(* Logix 5000 project; controller ProyectoIntegrador Emulate 5570 rev 30.12; software revision 30.00 *)

TASK MainTask (continuous, watchdog 500 ms) : MainProgram

MODULES
   Local : Emulate 5570 (ICP 2, rev 30.12)
      IO_module : vendor 1 type 0 code 15 (ICP 3, rev 1.1, Output RPI 150 ms)
END_MODULES

PROGRAM MainProgram   (* main routine MainRoutine *)
VAR
   Action_000 : SFC_ACTION := (Status := 16#0020_0000, PauseTimer := 1);
   Action_001 : SFC_ACTION := (Status := 16#0020_0000, PauseTimer := 1);
   Action_002 : SFC_ACTION := (Status := 16#0020_0000, PauseTimer := 1);
   Action_003 : SFC_ACTION := (Status := 16#0020_0000, PauseTimer := 1);
   Action_004 : SFC_ACTION := (Status := 16#0020_0000, PauseTimer := 1);
   Action_005 : SFC_ACTION := (Status := 16#0020_0000, PauseTimer := 1);
   Action_006 : SFC_ACTION := (Status := 16#0020_0000, PauseTimer := 1);
   Action_007 : SFC_ACTION := (Status := 16#0020_0000, PauseTimer := 1);
   Action_008 : SFC_ACTION := (Status := 16#0020_0000, PauseTimer := 1);
   Action_009 : SFC_ACTION := (Status := 16#0020_0000, PauseTimer := 1);
   Action_010 : SFC_ACTION := (Status := 16#0020_0000, PauseTimer := 1);
   Action_011 : SFC_ACTION := (Status := 16#0020_0000, PauseTimer := 1);
   Action_012 : SFC_ACTION := (Status := 16#0020_0000, PauseTimer := 1);
   Action_013 : SFC_ACTION := (Status := 16#0020_0000, PauseTimer := 1);
   Action_014 : SFC_ACTION := (Status := 16#0020_0000, PauseTimer := 1);
   Action_015 : SFC_ACTION := (Status := 16#0020_0000, PauseTimer := 1);
   Action_016 : SFC_ACTION := (Status := 16#0020_0000, PauseTimer := 1);
   Action_017 : SFC_ACTION := (Status := 16#0020_0000, PauseTimer := 1);
   Action_018 : SFC_ACTION := (Status := 16#0020_0000, PauseTimer := 1);
   Action_019 : SFC_ACTION := (Status := 16#0020_0000, PauseTimer := 1);
   Action_020 : SFC_ACTION := (Status := 16#0020_0000, PauseTimer := 1);
   Action_021 : SFC_ACTION := (Status := 16#0020_0000, PauseTimer := 1);
   Action_022 : SFC_ACTION := (Status := 16#0020_0000, PauseTimer := 1);
   Action_023 : SFC_ACTION := (Status := 16#0020_0000, PauseTimer := 1);
   Action_024 : SFC_ACTION := (Status := 16#0020_0000, PauseTimer := 1);
   Action_025 : SFC_ACTION := (Status := 16#0020_0000, PauseTimer := 1);
   Action_026 : SFC_ACTION := (Status := 16#0020_0000, PauseTimer := 1);
   Action_027 : SFC_ACTION := (Status := 16#0020_0000, PauseTimer := 1);
   Action_028 : SFC_ACTION := (Status := 16#0020_0000, PauseTimer := 1);
   Action_029 : SFC_ACTION := (Status := 16#0020_0000, PauseTimer := 1);
   BC_1 : BOOL;   // Encender/Apagar conveyor belt 1
   BC_2 : BOOL;   // Encender/Apagar conveyor belt 2
   BC_3 : BOOL;   // Encender/Apagar conveyor belt 3
   C1b : BOOL;   // Moves Cilinder 1 backward
   C1f : BOOL;   // Move cilinder 1 forward
   C2b : DINT;   // Move the cilinder 2 backwards
   C2f : BOOL;   // Move the cilinder 2 forward
   Cinta_gra : BOOL;   // El robot ya pegado en las cajas de la cinta grande
   Cinta_med : BOOL;   // El robot ya pegado en las cajas de la cinta media
   CintaRob : BOOL;   // El robot ya pegado en las cajas de la cinta pequena
   Clasif : BOOL;   // Encender/Apagar Classificador
   Compressor : BOOL;   // Encender/Apagar Compressor
   cont1 : COUNTER := (PRE := 3);
   cont2 : COUNTER := (PRE := 3);
   cont3 : COUNTER := (PRE := 3);
   cont4 : COUNTER := (PRE := 3);
   cont5 : COUNTER := (PRE := 3);
   cont6 : COUNTER := (PRE := 3);
   isBlue : BOOL;   // If the color detector in front of cilinder 1 detects blue color
   isGreen : BOOL;   // If the color detector in front of cilinder 1 detects green color
   isRed : BOOL;   // Normal or Color sensor for big boxes
   K1 : BOOL;   // Move la banda trasnportadora para esquerda y para trás
   K2 : BOOL;   // Move la banda transportadora para la direcha y para adelante
   K3 : BOOL;   // Move la banda trasnportadora para esquerda y para trás
   K4 : BOOL;   // Move la banda transportadora para la direcha y para adelante
   K5 : BOOL;   // Move la banda trasnportadora para esquerda y para trás
   K6 : BOOL;   // Move la banda transportadora para la direcha y para adelante
   Lavdo : BOOL;   // Encender/Apagar Lavado
   lConv : BOOL;   // Sensor de cajas conveyor belt 3 (vegetal grande)
   lCount : DINT;   // Large box counter
   mConv : BOOL;
   mCount : DINT;   // Medium Boxes count
   RC5 : BOOL;   // Encender/Apagar roller conveyor 4
   RC_1 : BOOL;   // Encender/Apagar roller conveyor 1
   RC_2 : BOOL;   // Encender/Apagar roller conveyor 2
   RC_3 : BOOL;   // Encender/Apagar roller conveyor 3
   RC_4 : BOOL;   // Encender/Apagar roller conveyor 4
   robotReady_L : BOOL;   // Un nível esta listo en la banda de cajas grandes
   robotReady_M : BOOL;   // Un nível esta listo en la banda de cajas medias
   robotReady_S : BOOL;   // Un nível esta listo en la banda de cajas pequenas
   S1_C1 : BOOL;   // Cilindro 1 recogido
   S1_C2 : BOOL;   // Sensor 1 final de carrera cilindro2
   S2_C1 : BOOL;   // Sensor 2 final de carrera cilindro 1
   S2_C2 : BOOL;   // Sensor 2 final de carrera cilindro 2
   S_clasif : DINT;   // Sensor para clasificacion de empaque
   sBC1 : BOOL;   // Tenemos una caja en el fin del tapete BC1
   sBC2 : BOOL;   // Tenemos una caja en el fin del tapete BC2
   sBC3 : BOOL;   // Tenemos una caja en el fin del tapete BC3
   sCount : DINT;   // Small Boxes Count
   Secado : BOOL;   // Encender/Apagar Secado
   Start : BOOL;   // Inicio del proceso
   Step_000 : SFC_STEP := (Status := 16#a820_0201, X := 1, SA := 1, DN := 1, PauseTimer := 1, T := 1176385, TMax := 1176385, Count := 1);
   Step_001 : SFC_STEP := (Status := 16#0020_0000, PauseTimer := 1);
   Step_002 : SFC_STEP := (Status := 16#0020_0000, PauseTimer := 1);
   Step_003 : SFC_STEP := (Status := 16#0020_0000, PauseTimer := 1);
   Step_004 : SFC_STEP := (Status := 16#0020_0000, PauseTimer := 1);
   Step_005 : SFC_STEP := (Status := 16#0020_0000, PauseTimer := 1);
   Step_006 : SFC_STEP := (Status := 16#0020_0000, PauseTimer := 1);
   Step_007 : SFC_STEP := (Status := 16#0020_0000, PauseTimer := 1);
   Step_008 : SFC_STEP := (Status := 16#0020_0000, PauseTimer := 1);
   Step_009 : SFC_STEP := (Status := 16#0020_0000, PauseTimer := 1);
   Step_010 : SFC_STEP := (Status := 16#0020_0000, PauseTimer := 1);
   Step_011 : SFC_STEP := (Status := 16#0020_0001, PauseTimer := 1);
   Step_012 : SFC_STEP := (Status := 16#0020_0001, PauseTimer := 1);
   Step_013 : SFC_STEP := (Status := 16#0020_0001, PauseTimer := 1);
   Step_014 : SFC_STEP := (Status := 16#0020_0001, PauseTimer := 1);
   Step_015 : SFC_STEP := (Status := 16#0020_0001, PauseTimer := 1);
   Step_016 : SFC_STEP := (Status := 16#0020_0000, PauseTimer := 1);
   Step_017 : SFC_STEP := (Status := 16#0020_0000, PauseTimer := 1);
   Step_018 : SFC_STEP := (Status := 16#0020_0000, PauseTimer := 1);
   Step_019 : SFC_STEP := (Status := 16#0020_0000, PauseTimer := 1);
   Step_020 : SFC_STEP := (Status := 16#0020_0000, PauseTimer := 1);
   Step_021 : SFC_STEP := (Status := 16#0020_0001, PauseTimer := 1);
   Step_022 : SFC_STEP := (Status := 16#0020_0001, PauseTimer := 1);
   Step_023 : SFC_STEP := (Status := 16#0020_0001, PauseTimer := 1);
   Step_024 : SFC_STEP := (Status := 16#0020_0001, PauseTimer := 1);
   Step_025 : SFC_STEP := (Status := 16#0020_0001, PauseTimer := 1);
   Step_026 : SFC_STEP := (Status := 16#0020_0000, PauseTimer := 1);
   Step_027 : SFC_STEP := (Status := 16#0020_0000, PauseTimer := 1);
   Step_028 : SFC_STEP := (Status := 16#0020_0000, PauseTimer := 1);
   Step_029 : SFC_STEP := (Status := 16#0020_0000, PauseTimer := 1);
   Step_030 : SFC_STEP := (Status := 16#0020_0000, PauseTimer := 1);
   Step_031 : SFC_STEP := (Status := 16#0020_0001, PauseTimer := 1);
   Step_032 : SFC_STEP := (Status := 16#0020_0000, PauseTimer := 1);
   Step_033 : SFC_STEP := (Status := 16#0020_0000, PauseTimer := 1);
   Step_034 : SFC_STEP := (Status := 16#0020_0000, PauseTimer := 1);
   Step_035 : SFC_STEP := (Status := 16#0020_0000, PauseTimer := 1);
   Step_036 : SFC_STEP := (Status := 16#0020_0000, PauseTimer := 1);
   Step_037 : SFC_STEP := (Status := 16#0020_0000, PauseTimer := 1);
   Step_038 : SFC_STEP := (Status := 16#0020_0000, PauseTimer := 1);
   Step_039 : SFC_STEP := (Status := 16#0020_0000, PauseTimer := 1);
   Step_041 : SFC_STEP := (Status := 16#0020_0001, PauseTimer := 1);
   Step_042 : SFC_STEP := (Status := 16#0020_0001, PauseTimer := 1);
   Step_100 : SFC_STEP := (Status := 16#0020_0000, PauseTimer := 1);
   Step_101 : SFC_STEP := (Status := 16#0020_0000, PauseTimer := 1);
   Step_102 : SFC_STEP := (Status := 16#0020_0000, PauseTimer := 1);
   Step_103 : SFC_STEP := (Status := 16#0020_0000, PauseTimer := 1);
   Step_200 : SFC_STEP := (Status := 16#0020_0000, PauseTimer := 1);   // Ligar la lógica de la clasificación y las alfombras correspondientes
   Step_201 : SFC_STEP := (Status := 16#0020_0000, PauseTimer := 1);
   Step_210 : SFC_STEP := (Status := 16#0020_0000, PauseTimer := 1);
   Step_211 : SFC_STEP := (Status := 16#0020_0000, PauseTimer := 1);
   Step_212 : SFC_STEP := (Status := 16#0020_0000, PauseTimer := 1);
   Step_213 : SFC_STEP := (Status := 16#0020_0000, PauseTimer := 1);
   Step_220 : SFC_STEP := (Status := 16#0020_0000, PauseTimer := 1);
   Step_221 : SFC_STEP := (Status := 16#0020_0000, PauseTimer := 1);
   Step_222 : SFC_STEP := (Status := 16#0020_0000, PauseTimer := 1);
   Step_223 : SFC_STEP := (Status := 16#0020_0000, PauseTimer := 1);
   Step_231 : SFC_STEP := (Status := 16#0020_0000, PauseTimer := 1);
   Stop : BOOL;   // Stop Button
   Stop_000 : SFC_STOP;
   Stop_001 : SFC_STOP;
   tCount : BOOL;   // Sensor de cajas en el volcador
   totalCount : DINT;   // Numero total de cjas
   Tran_000 : BOOL;
   Tran_001 : BOOL;
   Tran_002 : BOOL;
   Tran_003 : BOOL;
   Tran_004 : BOOL;
   Tran_005 : BOOL;
   Tran_006 : BOOL;
   Tran_007 : BOOL;
   Tran_008 : BOOL;
   Tran_009 : BOOL;
   Tran_010 : BOOL;
   Tran_011 : BOOL;
   Tran_012 : BOOL;
   Tran_013 : BOOL;
   Tran_014 : BOOL;
   Tran_015 : BOOL;
   Tran_016 : BOOL;
   Tran_017 : BOOL;
   Tran_018 : BOOL;
   Tran_019 : BOOL;
   Tran_020 : BOOL;
   Tran_021 : BOOL;
   Tran_022 : BOOL;
   Tran_023 : BOOL;
   Tran_024 : BOOL;
   Tran_025 : BOOL;
   Tran_026 : BOOL;
   Tran_027 : BOOL;
   Tran_028 : BOOL;
   Tran_029 : BOOL;
   Tran_030 : BOOL;
   Tran_031 : BOOL;
   Tran_032 : BOOL;
   Tran_033 : BOOL;
   Tran_034 : BOOL;
   Tran_035 : BOOL;
   Tran_036 : BOOL;
   Tran_037 : BOOL;
   Tran_038 : BOOL;
   Tran_039 : BOOL;
   Volcar : BOOL;   // Encendr/Apagar volcador
END_VAR

ROUTINE Distribution   (* sequential function chart *)
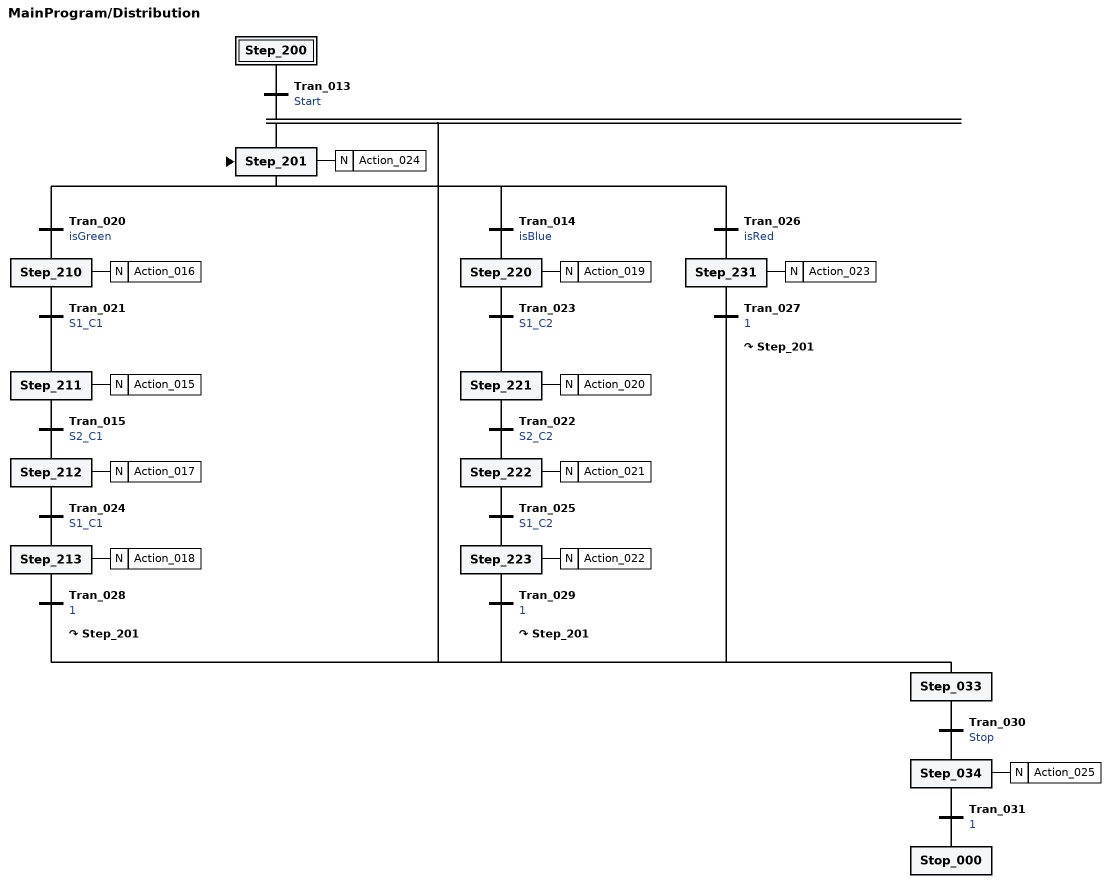
   // Small
   // Branch
   // Box Colors :
   // Green - Small
   // Blue - Medium
   // Red - Big
   // Big
   // Branch
   // Medium
   // Branch
   INITIAL_STEP Step_200:
   END_STEP
   TRANSITION Tran_013 FROM Step_200 TO (Step_201, Step_033)
      := Start
   END_TRANSITION
   STEP Step_201:
      ACTION Action_024 (N):
         RC5 := 1;
      END_ACTION
   END_STEP
   TRANSITION Tran_020 FROM Step_201 TO Step_210
      := isGreen
   END_TRANSITION
   STEP Step_033:
   END_STEP
   TRANSITION Tran_014 FROM Step_201 TO Step_220
      := isBlue
   END_TRANSITION
   TRANSITION Tran_026 FROM Step_201 TO Step_231
      := isRed
   END_TRANSITION
   STEP Step_210:
      ACTION Action_016 (N):
         RC5 := 0;
         (*If the cilinder isnt
         in its back position
         move it there *)
         IF not S1_C1 THEN
             C1b := 1;
         END_IF;
      END_ACTION
   END_STEP
   TRANSITION Tran_030 FROM Step_033 TO Step_034
      := Stop
         
   END_TRANSITION
   TRANSITION Tran_021 FROM Step_210 TO Step_211
      := S1_C1
   END_TRANSITION
   STEP Step_220:
      ACTION Action_019 (N):
         RC5 := 0;
         (*If the cilinder isnt
         in its back position
         move it there *)
         IF not S1_C2 THEN
             C2b := 1;
         END_IF;
      END_ACTION
   END_STEP
   STEP Step_231:
      ACTION Action_023 (N):
         //Jump back to the begining
         //Update the count
         lCount := lCount + 1 ;
      END_ACTION
   END_STEP
   STEP Step_034:
      ACTION Action_025 (N):
         RC5 := 0;
         C1f := 0;
         C2b := 0;
         C1b := 0;
         C2f := 0;
         
      END_ACTION
   END_STEP
   STEP Step_211:
      ACTION Action_015 (N):
         // Turn off cilinder 1 back
         C1b := 0;
         // Turn on cilinder 1 forward
         C1f := 1;
         
      END_ACTION
   END_STEP
   TRANSITION Tran_023 FROM Step_220 TO Step_221
      := S1_C2
   END_TRANSITION
   TRANSITION Tran_015 FROM Step_211 TO Step_212
      := S2_C1
   END_TRANSITION
   TRANSITION Tran_031 FROM Step_034 TO Stop_000
      := 1
         
   END_TRANSITION
   STEP Step_221:
      ACTION Action_020 (N):
         // Turn off cilinder 2 back
         C2b := 0;
         // Turn on cilinder 2 forward
         C2f := 1;
         
      END_ACTION
   END_STEP
   STEP Step_212:
      ACTION Action_017 (N):
         //Turn off cilinder 1 forward
         C1f:=0;
         // Turn on cilinder 1 back
         C1b:=1;
      END_ACTION
   END_STEP
   STOP Stop_000;
   TRANSITION Tran_022 FROM Step_221 TO Step_222
      := S2_C2
   END_TRANSITION
   TRANSITION Tran_024 FROM Step_212 TO Step_213
      := S1_C1
   END_TRANSITION
   STEP Step_222:
      ACTION Action_021 (N):
         //Turn off cilinder 1 forward
         C2f:=0;
         // Turn on cilinder 1 back
         C2b:=1;
      END_ACTION
   END_STEP
   STEP Step_213:
      ACTION Action_018 (N):
         //Turn off cilinder 1 back
         C1b:=0;
         //Jump back to the begining
         //Update the count
         sCount := sCount + 1 ;
      END_ACTION
   END_STEP
   TRANSITION Tran_025 FROM Step_222 TO Step_223
      := S1_C2
   END_TRANSITION
   STEP Step_223:
      ACTION Action_022 (N):
         //Turn off cilinder 1 back
         C2b:=0;
         //Jump back to the begining
         //Update the count
         mCount := mCount + 1 ;
      END_ACTION
   END_STEP
   TRANSITION Tran_028 FROM Step_213 TO (Step_201, Step_033)
      := 1
   END_TRANSITION
   TRANSITION Tran_027 FROM Step_231 TO (Step_201, Step_033)
      := 1
   END_TRANSITION
   TRANSITION Tran_029 FROM Step_223 TO (Step_201, Step_033)
      := 1
   END_TRANSITION
END_ROUTINE

ROUTINE Main   (* sequential function chart *)
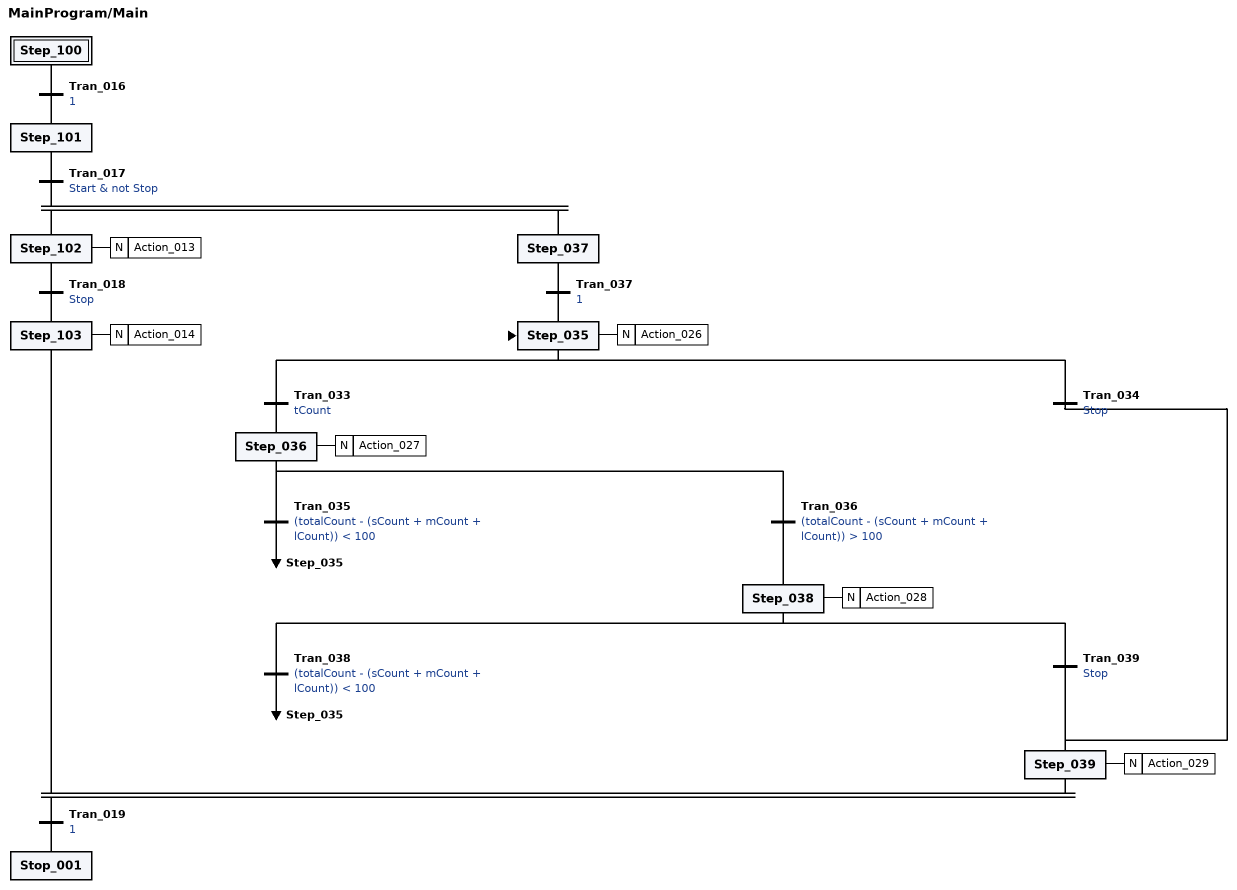
   // Change to
   // Rising Edge
   // - Look up
   // Guide
   // Change to
   // Rising Edge
   // - Look up
   // Guide
   // And with negative might help
   // but not perfect
   // When we reach at certain threshold we will
   // stop the admission of new boxes to the
   // system.
   INITIAL_STEP Step_100:
   END_STEP
   TRANSITION Tran_016 FROM Step_100 TO Step_101
      := 1
   END_TRANSITION
   STEP Step_101:
   END_STEP
   TRANSITION Tran_017 FROM Step_101 TO (Step_102, Step_037)
      := Start & not Stop
   END_TRANSITION
   STEP Step_102:
      ACTION Action_013 (N):
         RC_1 := 1;
         RC_2 := 1;
         RC_3 := 1;
         RC_4 := 1;
         Lavdo := 1;
         Secado := 1;
         Clasif := 1;
         Compressor := 1;
         //BC_1 := 1;
         //BC_2 := 1;
         //BC_3 := 1;
         
      END_ACTION
   END_STEP
   STEP Step_037:
   END_STEP
   TRANSITION Tran_037 FROM Step_037 TO Step_035
      := 1
   END_TRANSITION
   TRANSITION Tran_018 FROM Step_102 TO Step_103
      := Stop
   END_TRANSITION
   STEP Step_035:
      ACTION Action_026 (N):
         Volcar := 1;
      END_ACTION
   END_STEP
   STEP Step_103:
      ACTION Action_014 (N):
         RC_1 := 0;
         RC_2 := 0;
         RC_3 := 0;
         RC_4 := 0;
         Lavdo := 0;
         Secado := 0;
         Clasif := 0;
         Compressor := 0;
         BC_1 := 0;
         BC_2 := 0;
         BC_3 := 0;
         
      END_ACTION
   END_STEP
   TRANSITION Tran_033 FROM Step_035 TO Step_036
      := tCount
         
   END_TRANSITION
   STEP Step_036:
      ACTION Action_027 (N):
         totalCount := totalCount + 1 ;
      END_ACTION
   END_STEP
   TRANSITION Tran_035 FROM Step_036 TO Step_035
      := (totalCount - (sCount + mCount + lCount)) < 100
   END_TRANSITION
   TRANSITION Tran_036 FROM Step_036 TO Step_038
      := (totalCount - (sCount + mCount + lCount)) > 100
   END_TRANSITION
   STEP Step_038:
      ACTION Action_028 (N):
         Volcar := 0;
      END_ACTION
   END_STEP
   TRANSITION Tran_039 FROM Step_038 TO Step_039
      := Stop
         
   END_TRANSITION
   TRANSITION Tran_034 FROM Step_035 TO Step_039
      := Stop
   END_TRANSITION
   TRANSITION Tran_038 FROM Step_038 TO Step_035
      := (totalCount - (sCount + mCount + lCount)) < 100
   END_TRANSITION
   STEP Step_039:
      ACTION Action_029 (N):
         Volcar := 0;
      END_ACTION
   END_STEP
   TRANSITION Tran_019 FROM (Step_039, Step_103) TO Stop_001
      := 1
   END_TRANSITION
   STOP Stop_001;
END_ROUTINE

ROUTINE MainRoutine   (* ladder *)
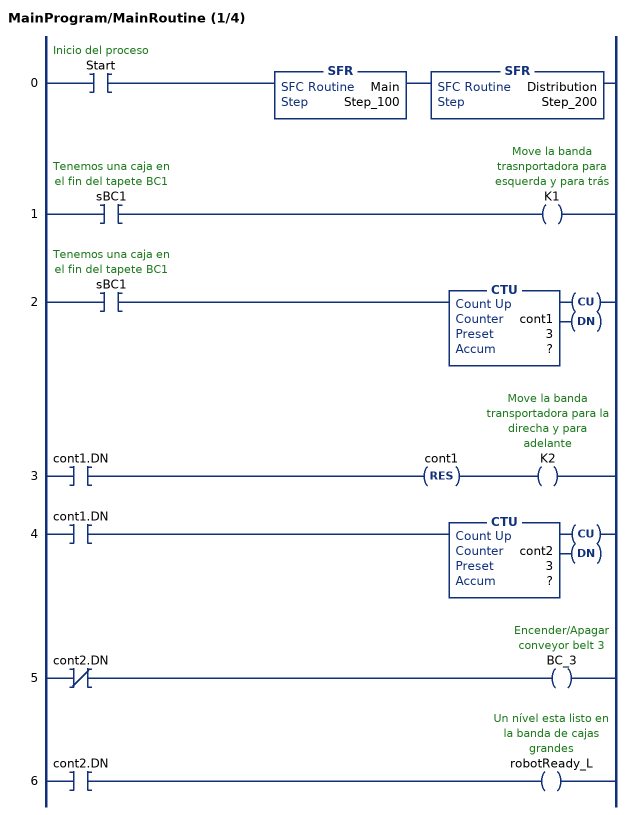
   0: XIC(Start)SFR(Main,Step_100)SFR(Distribution,Step_200);
   1: XIC(sBC1)OTE(K1);
   2: XIC(sBC1)CTU(cont1,?,?);
   3: XIC(cont1.DN)RES(cont1)OTE(K2);
   4: XIC(cont1.DN)CTU(cont2,?,?);
   5: XIO(cont2.DN)OTE(BC_3);
   6: XIC(cont2.DN)OTE(robotReady_L);
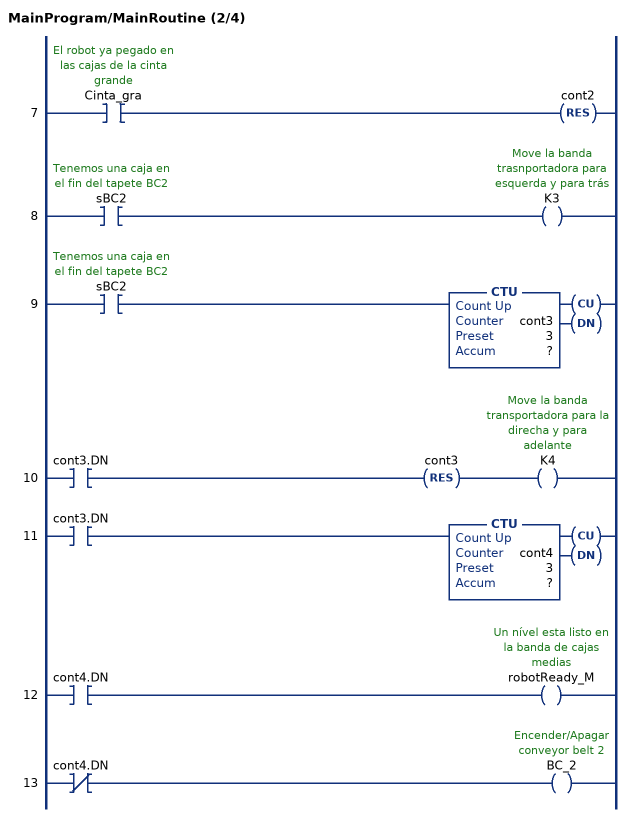
   7: XIC(Cinta_gra)RES(cont2);
   8: XIC(sBC2)OTE(K3);
   9: XIC(sBC2)CTU(cont3,?,?);
   10: XIC(cont3.DN)RES(cont3)OTE(K4);
   11: XIC(cont3.DN)CTU(cont4,?,?);
   12: XIC(cont4.DN)OTE(robotReady_M);
   13: XIO(cont4.DN)OTE(BC_2);
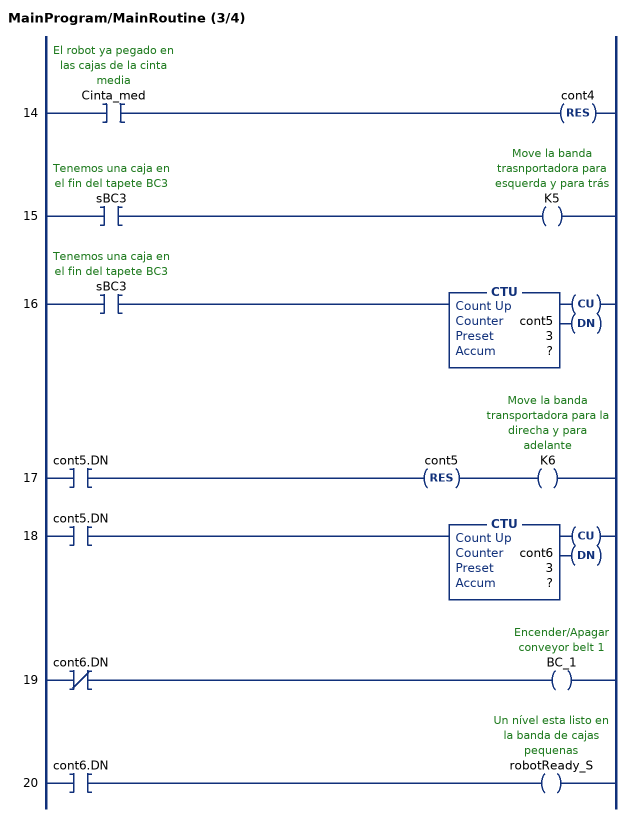
   14: XIC(Cinta_med)RES(cont4);
   15: XIC(sBC3)OTE(K5);
   16: XIC(sBC3)CTU(cont5,?,?);
   17: XIC(cont5.DN)RES(cont5)OTE(K6);
   18: XIC(cont5.DN)CTU(cont6,?,?);
   19: XIO(cont6.DN)OTE(BC_1);
   20: XIC(cont6.DN)OTE(robotReady_S);
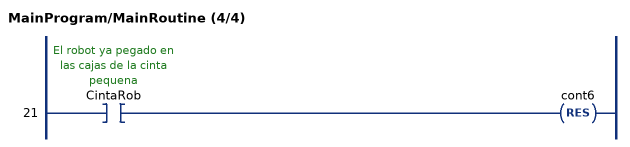
   21: XIC(CintaRob)RES(cont6);
END_ROUTINE
END_PROGRAM
